PROGRAM MAIN
VAR
    Estacion: FB_Estacion;
END_VAR

Estacion();

END_PROGRAM

(* stored: Version 1.1.0.1
   POU MAIN: Id {8e29b5fc-8f50-4b03-9cb8-d6b39838dd83}, SpecialFunc None *)
